TYPE Buttons :
STRUCT
	Start : BOOL;
	EStop : BOOL;
	Reset : BOOL;
END_STRUCT
END_TYPE

(* stored: Version 1.1.0.1, ProductVersion 3.1.4024.9
   DUT Buttons: Id {815586c7-3ac9-4ae9-bff2-6044bf00e4b0} *)
